(* IEC 61131-3 sources: SIGMATEK-Jumag-Utils-Examples/scaling/Class/Class0, 1 file *)

(* ---- Class0.st ---- *)
(*!
<Class
	Name               = "Class0"
	Revision           = "0.0"
	RealtimeTask       = "false"
	CyclicTask         = "true"
	DefCyclictime      = "100 ms"
	BackgroundTask     = "false"
	Sigmatek           = "false"
	OSInterface        = "false"
	HighPriority       = "false"
	Automatic          = "false"
	UpdateMode         = "Prescan"
	SharedCommandTable = "true"
	Objectsize         = "(284,120)">
	<Channels>
		<Server Name="ClassSvr" Visualized="false" Initialize="false" WriteProtected="true" Retentive="false"/>
		<Server Name="fScaled" Visualized="false" Initialize="false" WriteProtected="true" Retentive="false"/>
		<Server Name="iScaled" Visualized="false" Initialize="false" WriteProtected="true" Retentive="false"/>
		<Client Name="input" Required="true" Internal="false"/>
	</Channels>
	<Dependencies>
		<Files>
			<File Path=".\Source\scaling.c"/>
		</Files>
	</Dependencies>
</Class>
*)
Class0 : CLASS
  //Servers:
	ClassSvr 	: SvrChCmd_DINT;
	iScaled 	: SvrCh_DINT;
	fScaled 	: SvrCh_REAL;
  //Clients:
	input 	: CltCh_DINT;
  //Variables:
  //Functions:

	FUNCTION VIRTUAL GLOBAL CyWork
		VAR_INPUT
			EAX 	: UDINT;
		END_VAR
		VAR_OUTPUT
			state (EAX) 	: UDINT;
		END_VAR;
  //Tables:
	FUNCTION @STD
		VAR_OUTPUT
			ret_code	: CONFSTATES;
		END_VAR;
	FUNCTION GLOBAL TAB @CT_;
END_CLASS;

Function Global __cdecl map
VAR_INPUT
  INPUT : DINT;
  I_LO : DINT;
  I_HI : DINT;
  O_LO : DINT;
  O_HI : DINT;
END_VAR
VAR_OUTPUT
  Q : DINT;
END_VAR;

Function Global __cdecl fMap
VAR_INPUT
  INPUT : REAL;
  I_LO : REAL;
  I_HI : REAL;
  O_LO : REAL;
  O_HI : REAL;
END_VAR
VAR_OUTPUT
  Q : REAL;
END_VAR;

FUNCTION VIRTUAL GLOBAL Class0::CyWork
	VAR_INPUT
		EAX 	: UDINT;
	END_VAR
	VAR_OUTPUT
		state (EAX) 	: UDINT;
	END_VAR

  input := input.Read();

  iScaled := map(INPUT:= input, i_LO:= -200, I_HI:=200, O_LO:= 0, O_HI:= 100);
  fScaled := fMap(INPUT:= TO_REAL(input), I_LO:= TO_REAL(-200), I_HI:= TO_REAL(200), O_LO:= 0.0, O_HI:= 1000.0);

	state := READY;

END_FUNCTION
